FUNCTION_BLOCK Motor
VAR_INPUT
	//Software
	Stopped : BOOL;
	TurningClockwise : BOOL;
	TurningCounterclockwise : BOOL;
END_VAR
VAR_OUTPUT	
	AI_Position AT %I*: UINT;
	AI_Speed AT %I*: UDINT;
END_VAR
VAR	
	//Hardware
	DO_TurnClockwise AT %Q* : BOOL;
	DO_TurnCounterclockwise AT %Q* : BOOL;	
END_VAR

ACTION ACT_Stop:
DO_TurnClockwise := FALSE;
DO_TurnCounterclockwise := FALSE;

Stopped := TRUE;
TurningClockwise := FALSE;
TurningCounterclockwise := FALSE;
END_ACTION

ACTION ACT_TurnClockwise:
DO_TurnClockwise := TRUE;
DO_TurnCounterclockwise := FALSE;

Stopped := FALSE;
TurningClockwise := TRUE;
TurningCounterclockwise := FALSE;
END_ACTION

ACTION ACT_TurnCounterclockwise:
DO_TurnClockwise := FALSE;
DO_TurnCounterclockwise := TRUE;

Stopped := FALSE;
TurningClockwise := FALSE;
TurningCounterclockwise := TRUE;
END_ACTION

END_FUNCTION_BLOCK

(* stored: Version 1.1.0.1
   POU Motor: Id {55621e01-5c77-4d61-8dba-c3deb7c56a91}, SpecialFunc None
   Action ACT_Stop: Id {b2d47d70-1375-4b6a-869a-bd337a0d4ce1}
   Action ACT_TurnClockwise: Id {3e368d60-c229-49b8-82cd-74c2317d6232}
   Action ACT_TurnCounterclockwise: Id {b71b975d-7c90-43fc-80f5-f1fe34053cbc} *)
